// Mitsubishi GX Works2 project: 13. timer+counter+sequence_2   PLC: Q03UDV

PROGRAM MAIN
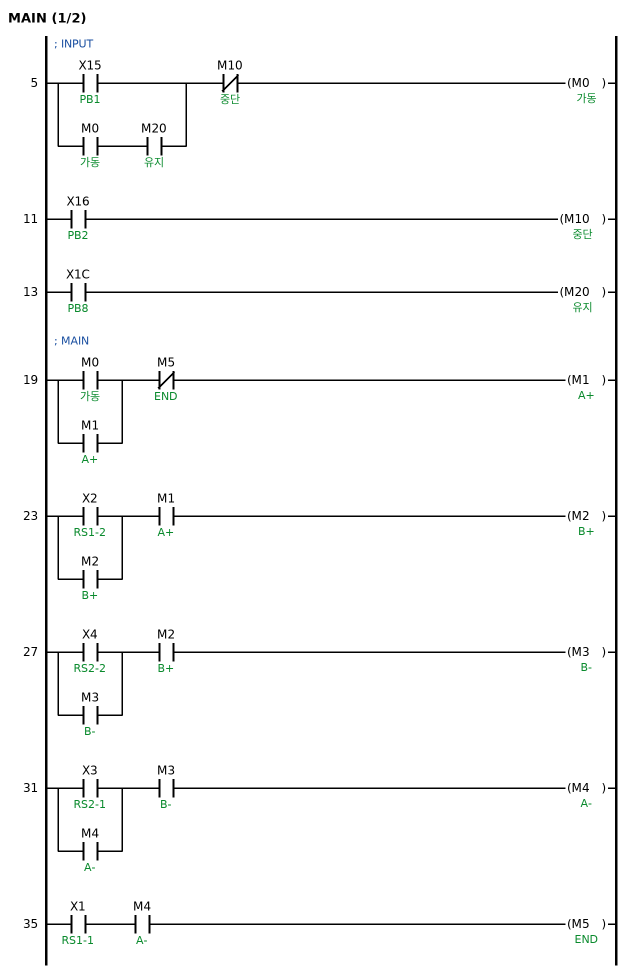
; INPUT
5     LD      X15  ; PB1
      LD      M0  ; 가동
      AND     M20  ; 유지
      ORB
      ANI     M10  ; 중단
      OUT     M0  ; 가동
11    LD      X16  ; PB2
      OUT     M10  ; 중단
13    LD      X1C  ; PB8
      OUT     M20  ; 유지
; MAIN
19    LD      M0  ; 가동
      OR      M1  ; A+
      ANI     M5  ; END
      OUT     M1  ; A+
23    LD      X2  ; RS1-2
      OR      M2  ; B+
      AND     M1  ; A+
      OUT     M2  ; B+
27    LD      X4  ; RS2-2
      OR      M3  ; B-
      AND     M2  ; B+
      OUT     M3  ; B-
31    LD      X3  ; RS2-1
      OR      M4  ; A-
      AND     M3  ; B-
      OUT     M4  ; A-
35    LD      X1  ; RS1-1
      AND     M4  ; A-
      OUT     M5  ; END
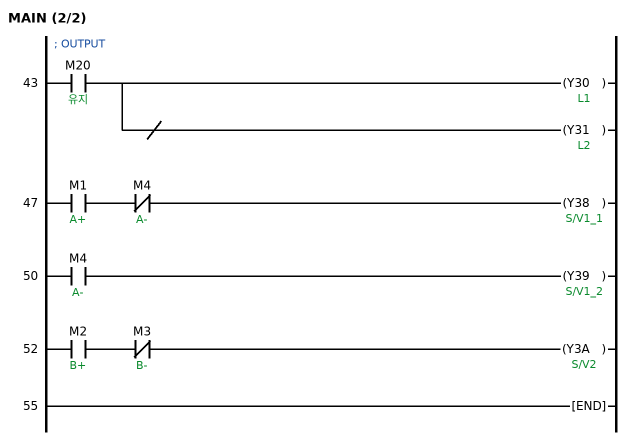
; OUTPUT
43    LD      M20  ; 유지
      OUT     Y30  ; L1
      INV
      OUT     Y31  ; L2
47    LD      M1  ; A+
      ANI     M4  ; A-
      OUT     Y38  ; S/V1_1
50    LD      M4  ; A-
      OUT     Y39  ; S/V1_2
52    LD      M2  ; B+
      ANI     M3  ; B-
      OUT     Y3A  ; S/V2
55    END
END_PROGRAM

// device comments not shown above
X17  ; PB3
X18  ; PB4
X19  ; PB5
X1A  ; PB6
X1B  ; PB7
M11  ; A+
M12  ; A-
M14  ; B+
M15  ; B-
M21  ; B+
M22  ; B-
M24  ; A+
M25  ; A-
Y32  ; L3
Y33  ; L4
Y34  ; L5
Y35  ; L6
Y36  ; L7
Y37  ; Buzzer
Y3B  ; S/V3
